PROGRAM INTERNAL P_EnumeratorExample
VAR
	bStart				: BOOL;
	sValue				: STRING(255);
	dtTime				: DT :=  DT#2023-5-8-12:55:23;
	fbStringBuilder1,
	fbStringBuilder2	: FB_StringBuilder;
	ipEnumerator		: I_Enumerator;
END_VAR

IF bStart THEN
	bStart := FALSE;
	
	fbStringBuilder1
		.Clear()
		.Append('   I love cats.')
		.Append('The time is: ').AppendAny(dtTime).Append('.')
		.BTrim();
	
	ipEnumerator := fbStringBuilder1.GetEnumerator();
	WHILE ipEnumerator.Next() DO
		fbStringBuilder2.Append(ipEnumerator.Current);
		END_WHILE
		
	sValue := fbStringBuilder2.GetString();
	END_IF

END_PROGRAM

(* stored: Version 1.1.0.1, ProductVersion 3.1.4024.4
   POU P_EnumeratorExample: Id {b227b542-53a7-4513-abcd-f9f25dca4fa9}, SpecialFunc None *)
